TYPE DS_CsvErrorLog EXTENDS DS_CsvLog :
STRUCT
	udiErrorId	: UDINT;
	iCaseid		: INT;
END_STRUCT
END_TYPE

(* stored: Version 1.1.0.1, ProductVersion 3.1.4024.12
   DUT DS_CsvErrorLog: Id {5547d62c-d280-4f47-810e-31a34e3ce3cd} *)
